LIN {X 0,Y 22.491,Z 717.935,A -85,B 0,C 180,E1 -30710.379,E2 -30710.379} C_VEL
LIN {X 0,Y 28.058,Z 716.021,A -85,B 0,C 180,E1 -30738.714,E2 -30738.714} C_VEL
LIN {X 0,Y 35.745,Z 713.471,A -85,B 0,C 180,E1 -30752.222,E2 -30752.222} C_VEL
LIN {X 0,Y 44.735,Z 709.958,A -85,B 0,C 180,E1 -30760.492,E2 -30760.492} C_VEL
LIN {X 0,Y 54.362,Z 705.391,A -85,B 0,C 180,E1 -30765.835,E2 -30765.835} C_VEL
LIN {X 0,Y 64.342,Z 699.656,A -85,B 0,C 180,E1 -30769.429,E2 -30769.429} C_VEL
LIN {X 0,Y 74.53,Z 692.568,A -85,B 0,C 180,E1 -30771.931,E2 -30771.931} C_VEL
LIN {X 0,Y 84.857,Z 683.773,A -85,B 0,C 180,E1 -30773.635,E2 -30773.635} C_VEL
LIN {X 0,Y 93.51,Z 674.789,A -85,B 0,C 180,E1 -30774.759,E2 -30774.759} C_VEL
LIN {X 0,Y 101.334,Z 664.967,A -85,B 0,C 180,E1 -30775.523,E2 -30775.523} C_VEL
LIN {X 0,Y 108.037,Z 654.615,A -85,B 0,C 180,E1 -30776.194,E2 -30776.194} C_VEL
LIN {X 0,Y 114.225,Z 642.534,A -85,B 0,C 180,E1 -30776.678,E2 -30776.678} C_VEL
LIN {X 0,Y 119.166,Z 629.692,A -85,B 0,C 180,E1 -30777.068,E2 -30777.068} C_VEL
LIN {X 0,Y 121.007,Z 623.315,A -85,B 0,C 180,E1 -30777.541,E2 -30777.541} C_VEL
LIN {X 0,Y 121.233,Z 621.841,A -85,B 0,C 180,E1 -30778.753,E2 -30778.753} C_VEL
LIN {X 0,Y 121.23,Z 621.364,A -85,B 0,C 180,E1 -30780,E2 -30780} C_VEL
LIN {X 0,Y 121.119,Z 621.454,A -85,B 0,C 180,E1 -30782.079,E2 -30782.079} C_VEL
LIN {X 0,Y 120.885,Z 623.018,A -85,B 0,C 180,E1 -30785.781,E2 -30785.781} C_VEL
LIN {X 0,Y 116.448,Z 635.995,A -85,B 0,C 180,E1 -30786.689,E2 -30786.689} C_VEL
LIN {X 0,Y 111.015,Z 647.543,A -85,B 0,C 180,E1 -30787.598,E2 -30787.598} C_VEL
LIN {X 0,Y 104.832,Z 657.888,A -85,B 0,C 180,E1 -30788.575,E2 -30788.575} C_VEL
LIN {X 0,Y 97.225,Z 668.188,A -85,B 0,C 180,E1 -30789.98,E2 -30789.98} C_VEL
LIN {X 0,Y 89.683,Z 676.58,A -85,B 0,C 180,E1 -30791.611,E2 -30791.611} C_VEL
LIN {X 0,Y 81.393,Z 684.291,A -85,B 0,C 180,E1 -30793.742,E2 -30793.742} C_VEL
LIN {X 0,Y 71.382,Z 691.941,A -85,B 0,C 180,E1 -30796.771,E2 -30796.771} C_VEL
LIN {X 0,Y 60.343,Z 698.732,A -85,B 0,C 180,E1 -30801.296,E2 -30801.296} C_VEL
LIN {X 0,Y 51.049,Z 703.331,A -85,B 0,C 180,E1 -30806.511,E2 -30806.511} C_VEL
LIN {X 0,Y 42.189,Z 706.865,A -85,B 0,C 180,E1 -30813.603,E2 -30813.603} C_VEL
LIN {X 0,Y 36.76,Z 708.684,A -85,B 0,C 180,E1 -30820.118,E2 -30820.118} C_VEL
LIN {X 0,Y 32.437,Z 709.907,A -85,B 0,C 180,E1 -30828.161,E2 -30828.161} C_VEL
LIN {X 0,Y 28.63,Z 710.937,A -85,B 0,C 180,E1 -30836.419,E2 -30836.419} C_VEL
LIN {X 0,Y 22.199,Z 712.2,A -85,B 0,C 180,E1 -30853.398,E2 -30853.398} C_VEL
LIN {X 0,Y 18.926,Z 712.635,A -85,B 0,C 180,E1 -30873.838,E2 -30873.838} C_VEL
LIN {X 0,Y 19.153,Z 712.541,A -85,B 0,C 180,E1 -30891.783,E2 -30891.783} C_VEL
LIN {X 0,Y 19.867,Z 712.388,A -85,B 0,C 180,E1 -30897.198,E2 -30897.198} C_VEL
LIN {X 0,Y 27.189,Z 711.053,A -85,B 0,C 180,E1 -30920.844,E2 -30920.844} C_VEL
LIN {X 0,Y 32.664,Z 709.751,A -85,B 0,C 180,E1 -30929.385,E2 -30929.385} C_VEL
LIN {X 0,Y 41.918,Z 706.906,A -85,B 0,C 180,E1 -30937.238,E2 -30937.238} C_VEL
LIN {X 0,Y 51.593,Z 703.066,A -85,B 0,C 180,E1 -30942.462,E2 -30942.462} C_VEL
LIN {X 0,Y 61.786,Z 697.97,A -85,B 0,C 180,E1 -30946.527,E2 -30946.527} C_VEL
LIN {X 0,Y 71.529,Z 691.92,A -85,B 0,C 180,E1 -30949.269,E2 -30949.269} C_VEL
LIN {X 0,Y 81.713,Z 684.122,A -85,B 0,C 180,E1 -30951.522,E2 -30951.522} C_VEL
LIN {X 0,Y 91.955,Z 674.431,A -85,B 0,C 180,E1 -30953.489,E2 -30953.489} C_VEL
LIN {X 0,Y 99.688,Z 665.362,A -85,B 0,C 180,E1 -30954.736,E2 -30954.736} C_VEL
LIN {X 0,Y 107.633,Z 653.773,A -85,B 0,C 180,E1 -30955.699,E2 -30955.699} C_VEL
LIN {X 0,Y 113.339,Z 643.29,A -85,B 0,C 180,E1 -30956.489,E2 -30956.489} C_VEL
LIN {X 0,Y 118.286,Z 631.581,A -85,B 0,C 180,E1 -30957.101,E2 -30957.101} C_VEL
LIN {X 0,Y 118.947,Z 629.633,A -85,B 0,C 180,E1 -30957.196,E2 -30957.196} C_VEL
LIN {X 0,Y 119.23,Z 628.795,A -85,B 0,C 180,E1 -30957.426,E2 -30957.426} C_VEL
LIN {X 0,Y 119.407,Z 628.446,A -85,B 0,C 180,E1 -30959.119,E2 -30959.119} C_VEL
LIN {X 0,Y 118.853,Z 630.173,A -85,B 0,C 180,E1 -30959.514,E2 -30959.514} C_VEL
LIN {X 0,Y 114.114,Z 642.11,A -85,B 0,C 180,E1 -30959.74,E2 -30959.74} C_VEL
LIN {X 0,Y 107.841,Z 654.087,A -85,B 0,C 180,E1 -30960.052,E2 -30960.052} C_VEL
LIN {X 0,Y 100.15,Z 665.594,A -85,B 0,C 180,E1 -30960.509,E2 -30960.509} C_VEL
LIN {X 0,Y 91.376,Z 676.116,A -85,B 0,C 180,E1 -30961.001,E2 -30961.001} C_VEL
LIN {X 0,Y 82.613,Z 684.671,A -85,B 0,C 180,E1 -30961.703,E2 -30961.703} C_VEL
LIN {X 0,Y 72.121,Z 693.051,A -85,B 0,C 180,E1 -30962.791,E2 -30962.791} C_VEL
LIN {X 0,Y 61.689,Z 699.878,A -85,B 0,C 180,E1 -30964.56,E2 -30964.56} C_VEL
LIN {X 0,Y 49.654,Z 706.196,A -85,B 0,C 180,E1 -30967.802,E2 -30967.802} C_VEL
LIN {X 0,Y 39.542,Z 710.356,A -85,B 0,C 180,E1 -30972.174,E2 -30972.174} C_VEL
LIN {X 0,Y 29.844,Z 713.497,A -85,B 0,C 180,E1 -30979.621,E2 -30979.621} C_VEL
LIN {X 0,Y 18.917,Z 716.229,A -85,B 0,C 180,E1 -31002.009,E2 -31002.009} C_VEL
LIN {X 0,Y 15.715,Z 717.022,A -85,B 0,C 180,E1 -31023.435,E2 -31023.435} C_VEL
LIN {X 0,Y 15.376,Z 717.412,A -85,B 0,C 180,E1 -31050,E2 -31050} C_VEL
LIN {X 0,Y 15.787,Z 716.99,A -85,B 0,C 180,E1 -31077.084,E2 -31077.084} C_VEL
LIN {X 0,Y 23.948,Z 715.015,A -85,B 0,C 180,E1 -31111.689,E2 -31111.689} C_VEL
LIN {X 0,Y 33.02,Z 712.463,A -85,B 0,C 180,E1 -31123.29,E2 -31123.29} C_VEL
LIN {X 0,Y 42.881,Z 708.952,A -85,B 0,C 180,E1 -31129.531,E2 -31129.531} C_VEL
LIN {X 0,Y 53.065,Z 704.383,A -85,B 0,C 180,E1 -31133.353,E2 -31133.353} C_VEL
LIN {X 0,Y 63.423,Z 698.652,A -85,B 0,C 180,E1 -31135.768,E2 -31135.768} C_VEL
LIN {X 0,Y 73.868,Z 691.565,A -85,B 0,C 180,E1 -31137.409,E2 -31137.409} C_VEL
LIN {X 0,Y 84.365,Z 682.771,A -85,B 0,C 180,E1 -31138.437,E2 -31138.437} C_VEL
LIN {X 0,Y 93.13,Z 673.785,A -85,B 0,C 180,E1 -31139.124,E2 -31139.124} C_VEL
LIN {X 0,Y 101.028,Z 663.961,A -85,B 0,C 180,E1 -31139.554,E2 -31139.554} C_VEL
LIN {X 0,Y 108.43,Z 652.523,A -85,B 0,C 180,E1 -31139.977,E2 -31139.977} C_VEL
LIN {X 0,Y 114.749,Z 639.898,A -85,B 0,C 180,E1 -31140.292,E2 -31140.292} C_VEL
LIN {X 0,Y 118.904,Z 629.008,A -85,B 0,C 180,E1 -31140.5,E2 -31140.5} C_VEL
LIN {X 0,Y 119.194,Z 628.11,A -85,B 0,C 180,E1 -31140.665,E2 -31140.665} C_VEL
LIN {X 0,Y 118.961,Z 628.568,A -85,B 0,C 180,E1 -31142.583,E2 -31142.583} C_VEL
LIN {X 0,Y 117.761,Z 632.067,A -85,B 0,C 180,E1 -31142.953,E2 -31142.953} C_VEL
LIN {X 0,Y 112.67,Z 643.946,A -85,B 0,C 180,E1 -31143.622,E2 -31143.622} C_VEL
LIN {X 0,Y 107.05,Z 654.169,A -85,B 0,C 180,E1 -31144.369,E2 -31144.369} C_VEL
LIN {X 0,Y 99.702,Z 664.885,A -85,B 0,C 180,E1 -31145.347,E2 -31145.347} C_VEL
LIN {X 0,Y 91.963,Z 674.054,A -85,B 0,C 180,E1 -31146.554,E2 -31146.554} C_VEL
LIN {X 0,Y 83.421,Z 682.378,A -85,B 0,C 180,E1 -31148.155,E2 -31148.155} C_VEL
LIN {X 0,Y 73.229,Z 690.472,A -85,B 0,C 180,E1 -31150.358,E2 -31150.358} C_VEL
LIN {X 0,Y 62.148,Z 697.566,A -85,B 0,C 180,E1 -31153.393,E2 -31153.393} C_VEL
LIN {X 0,Y 51.601,Z 702.921,A -85,B 0,C 180,E1 -31157.566,E2 -31157.566} C_VEL
LIN {X 0,Y 41.921,Z 706.8,A -85,B 0,C 180,E1 -31162.772,E2 -31162.772} C_VEL
LIN {X 0,Y 32.676,Z 709.673,A -85,B 0,C 180,E1 -31170.648,E2 -31170.648} C_VEL
LIN {X 0,Y 22.513,Z 711.94,A -85,B 0,C 180,E1 -31191.367,E2 -31191.367} C_VEL
LIN {X 0,Y 17.72,Z 712.759,A -85,B 0,C 180,E1 -31230,E2 -31230} C_VEL
LIN {X 0,Y 19.867,Z 712.388,A -85,B 0,C 180,E1 -31257.198,E2 -31257.198} C_VEL
LIN {X 0,Y 21.29,Z 712.204,A -85,B 0,C 180,E1 -31267.57,E2 -31267.57} C_VEL
LIN {X 0,Y 23.393,Z 711.928,A -85,B 0,C 180,E1 -31284.151,E2 -31284.151} C_VEL
LIN {X 0,Y 26.994,Z 711.361,A -85,B 0,C 180,E1 -31297.188,E2 -31297.188} C_VEL
LIN {X 0,Y 30.246,Z 710.591,A -85,B 0,C 180,E1 -31301.541,E2 -31301.541} C_VEL
LIN {X 0,Y 43.095,Z 706.723,A -85,B 0,C 180,E1 -31308.089,E2 -31308.089} C_VEL
LIN {X 0,Y 53.341,Z 702.521,A -85,B 0,C 180,E1 -31311.167,E2 -31311.167} C_VEL
LIN {X 0,Y 65.366,Z 696.206,A -85,B 0,C 180,E1 -31313.999,E2 -31313.999} C_VEL
LIN {X 0,Y 75.764,Z 689.216,A -85,B 0,C 180,E1 -31315.682,E2 -31315.682} C_VEL
LIN {X 0,Y 77.499,Z 687.896,A -85,B 0,C 180,E1 -31315.955,E2 -31315.955} C_VEL
LIN {X 0,Y 77.419,Z 688.077,A -85,B 0,C 180,E1 -31316.911,E2 -31316.911} C_VEL
LIN {X 0,Y 66.828,Z 695.644,A -85,B 0,C 180,E1 -31317.49,E2 -31317.49} C_VEL
LIN {X 0,Y 56.242,Z 701.779,A -85,B 0,C 180,E1 -31318.482,E2 -31318.482} C_VEL
LIN {X 0,Y 46.572,Z 706.312,A -85,B 0,C 180,E1 -31320,E2 -31320} C_VEL
LIN {X 0,Y 35.182,Z 710.493,A -85,B 0,C 180,E1 -31322.842,E2 -31322.842} C_VEL
LIN {X 0,Y 28.256,Z 712.49,A -85,B 0,C 180,E1 -31325.802,E2 -31325.802} C_VEL
LIN {X 0,Y 15.088,Z 715.22,A -85,B 0,C 180,E1 -31341.317,E2 -31341.317} C_VEL
LIN {X 0,Y 9.4,Z 716.088,A -85,B 0,C 180,E1 -31368.385,E2 -31368.385} C_VEL
LIN {X 0,Y 8.228,Z 716.407,A -85,B 0,C 180,E1 -31410,E2 -31410} C_VEL
LIN {X 0,Y 9.867,Z 715.998,A -85,B 0,C 180,E1 -31455.418,E2 -31455.418} C_VEL
LIN {X 0,Y 21.496,Z 714.007,A -85,B 0,C 180,E1 -31488.751,E2 -31488.751} C_VEL
LIN {X 0,Y 31.712,Z 711.456,A -85,B 0,C 180,E1 -31495.767,E2 -31495.767} C_VEL
LIN {X 0,Y 42.172,Z 707.947,A -85,B 0,C 180,E1 -31499.12,E2 -31499.12} C_VEL
LIN {X 0,Y 52.718,Z 703.377,A -85,B 0,C 180,E1 -31501.093,E2 -31501.093} C_VEL
LIN {X 0,Y 64.883,Z 696.704,A -85,B 0,C 180,E1 -31502.305,E2 -31502.305} C_VEL
LIN {X 0,Y 75.654,Z 689.199,A -85,B 0,C 180,E1 -31503.021,E2 -31503.021} C_VEL
LIN {X 0,Y 77.418,Z 687.822,A -85,B 0,C 180,E1 -31503.079,E2 -31503.079} C_VEL
LIN {X 0,Y 77.5,Z 687.636,A -85,B 0,C 180,E1 -31504.052,E2 -31504.052} C_VEL
LIN {X 0,Y 67.104,Z 694.896,A -85,B 0,C 180,E1 -31505.767,E2 -31505.767} C_VEL
LIN {X 0,Y 56.769,Z 700.711,A -85,B 0,C 180,E1 -31507.958,E2 -31507.958} C_VEL
LIN {X 0,Y 46.508,Z 705.309,A -85,B 0,C 180,E1 -31510.82,E2 -31510.82} C_VEL
LIN {X 0,Y 36.346,Z 708.844,A -85,B 0,C 180,E1 -31514.808,E2 -31514.808} C_VEL
LIN {X 0,Y 29.714,Z 710.662,A -85,B 0,C 180,E1 -31518.904,E2 -31518.904} C_VEL
LIN {X 0,Y 17.579,Z 712.929,A -85,B 0,C 180,E1 -31536.912,E2 -31536.912} C_VEL
LIN {X 0,Y 10.692,Z 713.747,A -85,B 0,C 180,E1 -31590,E2 -31590} C_VEL
LIN {X 0,Y 17.577,Z 712.966,A -85,B 0,C 180,E1 -31643.098,E2 -31643.098} C_VEL
LIN {X 0,Y 29.707,Z 710.739,A -85,B 0,C 180,E1 -31661.137,E2 -31661.137} C_VEL
LIN {X 0,Y 30.246,Z 710.591,A -85,B 0,C 180,E1 -31661.541,E2 -31661.541} C_VEL
LIN {X 0,Y 29.831,Z 710.778,A -85,B 0,C 180,E1 -31663.324,E2 -31663.324} C_VEL
LIN {X 0,Y 26.049,Z 711.831,A -85,B 0,C 180,E1 -31666.59,E2 -31666.59} C_VEL
LIN {X 0,Y 17.438,Z 713.683,A -85,B 0,C 180,E1 -31670.626,E2 -31670.626} C_VEL
LIN {X 0,Y 9.769,Z 714.701,A -85,B 0,C 180,E1 -31675.178,E2 -31675.178} C_VEL
LIN {X 0,Y 1.08,Z 715.402,A -85,B 0,C 180,E1 -31770,E2 -31770} C_VEL
LIN {X 0,Y 7.032,Z 714.99,A -85,B 0,C 180,E1 -31861.97,E2 -31861.97} C_VEL
LIN {X 0,Y 21.293,Z 712.998,A -85,B 0,C 180,E1 -31868.045,E2 -31868.045} C_VEL
LIN {X 0,Y 14.492,Z 713.917,A -85,B 0,C 180,E1 -31874.096,E2 -31874.096} C_VEL
LIN {X 0,Y 3.664,Z 714.735,A -85,B 0,C 180,E1 -31950,E2 -31950} C_VEL
LIN {X 0,Y 14.491,Z 713.954,A -85,B 0,C 180,E1 -32025.919,E2 -32025.919} C_VEL
LIN {X 0,Y 21.298,Z 713.042,A -85,B 0,C 180,E1 -32031.855,E2 -32031.855} C_VEL
LIN {X 0,Y 9.769,Z 714.701,A -85,B 0,C 180,E1 -32035.178,E2 -32035.178} C_VEL
LIN {X 0,Y 9.769,Z 714.701,A -85,B 0,C 180,E1 -32035.178,E2 -32035.178}

QRS_NEXT_CUT()

QRS_NEXT()
QRS_HOME()

END
